// TwinCAT 3 PLC project TcToolkitSample_PLC
// ProgramVersion: 3.1.4026.22
// libraries:
//   TwinCat Dynamic Collections, * (FisoThemes)
//   Tc2_Standard, * (Beckhoff Automation GmbH)
//   Tc2_System, * (Beckhoff Automation GmbH)
// project tree:
//   / PlcTask.TcTTO
//   POUs/ MAIN.TcPOU, P_Startup.TcPOU, F_Scale.TcPOU
//   DUTs/ E_StationState.TcDUT, E_Command.TcDUT, ST_Status.TcDUT (not stored), ST_StationStatus.TcDUT, ST_Recipe.TcDUT (not stored), U_Word.TcDUT, T_Ident.TcDUT
//   GVLs/ GVL_Io.TcGVL (not stored), GVL_System.TcGVL, GVL_Hmi.TcGVL
//   POUs/Interfaces/ I_Resettable.TcIO (not stored), I_Diagnosable.TcIO, I_Station.TcIO (not stored)
//   POUs/Actuators/ FB_Cylinder.TcPOU
//   POUs/Machine/ FB_Station.TcPOU, FB_StationDerived.TcPOU (not stored)
// real-time tasks:
//   TASK PlcTask: cycle T#10ms, priority 20, ADS port 350

CONFIGURATION TcToolkitSample_PLC
    RESOURCE PLC ON TwinCAT3
        TASK PlcTask(INTERVAL := T#10ms, PRIORITY := 20);
        PROGRAM MAIN WITH PlcTask : MAIN;
    END_RESOURCE
END_CONFIGURATION

// ---- DUTs/E_StationState.TcDUT
TYPE E_StationState :
(
	Idle := 0,
	Running := 1,
	Error := 2,
	Done := 3
) DINT;
END_TYPE

// ---- DUTs/E_Command.TcDUT
TYPE E_Command :
(
	None,
	Start,
	Stop,
	Reset
);
END_TYPE

// ---- DUTs/ST_StationStatus.TcDUT
TYPE ST_StationStatus EXTENDS ST_Status :
STRUCT
	eState	: E_StationState;
	sName	: STRING(31);
END_STRUCT
END_TYPE

// ---- DUTs/U_Word.TcDUT
TYPE U_Word :
UNION
	nWord	: WORD;
	aBytes	: ARRAY[0..1] OF BYTE;
END_UNION
END_TYPE

// ---- DUTs/T_Ident.TcDUT
TYPE T_Ident : STRING(31);
END_TYPE

// ---- GVLs/GVL_System.TcGVL
{attribute 'qualified_only'}
VAR_GLOBAL
	fbCylinder	: FB_Cylinder(refExtendOut := GVL_Io.bExtendOut, refRetractOut := GVL_Io.bRetractOut);
	fbStation	: FB_Station;
	fbDerived	: FB_StationDerived;
END_VAR

// ---- GVLs/GVL_Hmi.TcGVL
{attribute 'qualified_only'}
VAR_GLOBAL
	nSpeed		: INT;
	bEnable		: BOOL;
	arValues	: ARRAY[0..9] OF INT;
END_VAR

// ---- POUs/Interfaces/I_Diagnosable.TcIO
INTERFACE I_Diagnosable

PROPERTY ErrorId : UDINT
GET
END_GET
END_PROPERTY

END_INTERFACE

// ---- POUs/MAIN.TcPOU
PROGRAM MAIN
VAR
	nCycleCount	: UDINT;
	nIdx		: INT;
	fScaled		: LREAL;
END_VAR

nCycleCount := nCycleCount + 1;

GVL_System.fbCylinder.Cyclic();
GVL_System.fbStation.Cyclic();
GVL_System.fbDerived.Cyclic();

GVL_Hmi.bEnable := (GVL_System.fbStation.State = E_StationState.Running);

fScaled := F_Scale(fValue := 5.0, fMin := 0.0, fMax := 10.0);
GVL_Hmi.nSpeed := LREAL_TO_INT(fScaled * 100.0);

FOR nIdx := 0 TO 9 DO
	GVL_Hmi.arValues[nIdx] := GVL_Hmi.nSpeed;
END_FOR

END_PROGRAM

// ---- POUs/F_Scale.TcPOU
FUNCTION F_Scale : LREAL
VAR_INPUT
	fValue, fMin, fMax	: LREAL;
END_VAR
VAR
	fSpan	: LREAL;
END_VAR

fSpan := fMax - fMin;

IF fSpan = 0 THEN
	F_Scale := 0;
ELSE
	F_Scale := (fValue - fMin) / fSpan;
END_IF

END_FUNCTION

// ---- POUs/Actuators/FB_Cylinder.TcPOU
FUNCTION_BLOCK FB_Cylinder
VAR
	_bExtended, _bRetracted	: BOOL;
	refExtendOut			: REFERENCE TO BOOL;
	refRetractOut			: REFERENCE TO BOOL;
END_VAR

// The cylinder is edge-free: the sensor image is refreshed every cycle and the outputs
// are held by whichever of Extend()/Retract() was called last.
Cyclic();

METHOD FB_init : BOOL
VAR_INPUT
	bInitRetains	: BOOL;
	bInCopyCode		: BOOL;
	refExtendOut	: REFERENCE TO BOOL;
	refRetractOut	: REFERENCE TO BOOL;
END_VAR
THIS^.refExtendOut REF= refExtendOut;
THIS^.refRetractOut REF= refRetractOut;
FB_init := TRUE;
END_METHOD

METHOD Extend : BOOL
VAR
END_VAR
refExtendOut := TRUE;
refRetractOut := FALSE;
Extend := TRUE;
END_METHOD

METHOD Retract : BOOL
VAR
END_VAR
refExtendOut := FALSE;
refRetractOut := TRUE;
Retract := TRUE;
END_METHOD

METHOD Cyclic
VAR
END_VAR
_bExtended := GVL_Io.bSensorExtended;
_bRetracted := GVL_Io.bSensorRetracted;
END_METHOD

PROPERTY bIsExtended : BOOL
GET
bIsExtended := _bExtended;
END_GET
END_PROPERTY

PROPERTY bIsRetracted : BOOL
GET
bIsRetracted := _bRetracted;
END_GET
END_PROPERTY

END_FUNCTION_BLOCK

// ---- POUs/Machine/FB_Station.TcPOU
FUNCTION_BLOCK FB_Station IMPLEMENTS I_Station
VAR
	refCylinder	: REFERENCE TO FB_Cylinder;
	_eState		: E_StationState;
	_eCommand	: E_Command;
	_stStatus	: ST_StationStatus;
	_stRecipe	: ST_Recipe;
	_uWord		: U_Word;
	_sIdent		: T_Ident;
	_nErrorId	: UDINT;
END_VAR

Cyclic();

METHOD Cyclic
VAR
	bExtended	: BOOL;
END_VAR
bExtended := refCylinder.bIsExtended;

CASE _eState OF
	E_StationState.Idle:
		IF _eCommand = E_Command.Start THEN
			_eState := E_StationState.Running;
		END_IF

	E_StationState.Running:
		IF bExtended THEN
			refCylinder.Retract();
		ELSE
			refCylinder.Extend();
		END_IF
		IF _nErrorId <> 0 THEN
			_eState := E_StationState.Error;
		END_IF

	E_StationState.Error:
		_stStatus.bError := TRUE;

	E_StationState.Done:
		_stStatus.bDone := TRUE;
END_CASE

_stStatus.eState := _eState;
_stStatus.nErrorId := _nErrorId;
_uWord.nWord := _stRecipe.aSteps[1];
END_METHOD

METHOD Execute : BOOL
VAR
END_VAR
IF _eState = E_StationState.Idle THEN
	_eCommand := E_Command.Start;
	_stStatus.bBusy := TRUE;
	Execute := TRUE;
ELSE
	Execute := FALSE;
END_IF
END_METHOD

METHOD Reset : BOOL
VAR
END_VAR
_eState := E_StationState.Idle;
_eCommand := E_Command.None;
_nErrorId := 0;
_stStatus.bBusy := FALSE;
_stStatus.bDone := FALSE;
_stStatus.bError := FALSE;
_stStatus.nErrorId := 0;
Reset := TRUE;
END_METHOD

PROPERTY State : E_StationState
GET
State := _eState;
END_GET
SET
_eState := State;
END_SET
END_PROPERTY

PROPERTY ErrorId : UDINT
GET
ErrorId := _nErrorId;
END_GET
END_PROPERTY

ACTION Act_Home:
refCylinder REF= GVL_System.fbCylinder;
refCylinder.Retract();
_eState := E_StationState.Idle;
_sIdent := 'STATION-01';
END_ACTION

END_FUNCTION_BLOCK

// ---- POUs/P_Startup.TcPOU
PROGRAM P_Startup
VAR
	bDone	: BOOL;
END_VAR

IF NOT bDone THEN
	GVL_System.fbStation.Reset();
	GVL_System.fbDerived.Reset();
	GVL_Hmi.nSpeed := 50;
	bDone := TRUE;
END_IF

END_PROGRAM
